Universal Robots PolyScope program: TurnToolFlange.urp

ProgramRoot directory=/home/ur/ursim-3.1/programs; kinematics=(a=[0, -0.425, -0.39225, 0, 0, 0], d=[0.08916, 0, 0, 0.10915, 0.09465, 0.0823], alpha=[1.5708, 0, 0, 1.5708, -1.5708, 0], deltaTheta=[0, 0, 0, 0, 0, 0], status=notInitialized); lastSavedInVersion=(project__name=Polyscope, major__version=3, minor__version=1, svn__revision=17195, build__date=Mar 11 2015, 13:02:28); name=TurnToolFlange; programVersion=(project__name=Polyscope, major__version=3, minor__version=1, svn__revision=17195, build__date=Mar 11 2015, 13:02:28); robotEnvironmentFileName=default; serialNumberRobot=2014350001
  MainProgram cartesianAcceleration=1.2; cartesianSpeed=0.25; jointAcceleration=1.3962634015954636; jointSpeed=1.0471975511965976; sharedProcessMoveBlendRadius=0.025; motionType=JOINT_SPACE; runOnlyOneCycle=true
    Move cartesianAcceleration=1.2; cartesianSpeed=0.25; jointAcceleration=1.3962634015954636; jointSpeed=1.0471975511965976; sharedProcessMoveBlendRadius=0.025; motionType=JOINT_SPACE
      Waypoint blendRadius=0.05; cartesianAcceleration=1.2; cartesianSpeed=0.25; jointAcceleration=1.3962634015954636; jointSpeed=1.0471975511965976; nextMotionTime=2.0; stoppoint=true; useSharedBlendParameter=true; useSharedParameters=true; outputFlangePose=(pos=(x=-0.12011316349511432, y=-0.4317629397815833, z=0.33440045381825007), rot=(x=-0.0012209830283371023, y=3.116276481240665, z=0.038891916168164946)); position=TCP in base x=-120.113 y=-431.763 z=334.4 mm, rx=-0.0012 ry=3.1163 rz=0.0389 rad; joints [-91.713, -84.826, -108.941, -77.706, 91.393, -1.776] deg; positionType=FIXED_POSITION; waypointPoseInFeatureCoordinates=(pos=(x=-0.12011316299633705, y=-0.4317629218220435, z=0.33440041081305716), rot=(x=-0.0012209830284087941, y=3.116276481240896, z=0.03889191616813282)); name=actual_pos
    Assignment expr=get_actual_joint_positions(); operatorValueType=INTEGER; valueSource=EXPRESSION
    Script type=0; expressionBranchNode=ExpressionVariableNode[5]=joint[5]+d2r(90)
    If checkConditionInSeperateThread=true; expr=ExpressionIONode≟ False; type=IF_NODE
      Move cartesianAcceleration=1.2; cartesianSpeed=0.25; jointAcceleration=1.3962634015954636; jointSpeed=1.0471975511965976; sharedProcessMoveBlendRadius=0.025; motionType=JOINT_SPACE
        Waypoint blendRadius=0.05; cartesianAcceleration=1.2; cartesianSpeed=0.25; jointAcceleration=1.3962634015954636; jointSpeed=1.0471975511965976; nextMotionTime=2.0; stoppoint=true; useSharedBlendParameter=true; useSharedParameters=true; positionType=VARIABLE_POSITION; name=Waypoint
    If type=ELSE_NODE
      Move cartesianAcceleration=1.2; cartesianSpeed=0.25; jointAcceleration=1.3962634015954636; jointSpeed=1.0471975511965976; sharedProcessMoveBlendRadius=0.025; motionType=JOINT_SPACE
        Waypoint blendRadius=0.05; cartesianAcceleration=1.2; cartesianSpeed=0.25; jointAcceleration=1.3962634015954636; jointSpeed=1.0471975511965976; nextMotionTime=2.0; stoppoint=true; useSharedBlendParameter=true; useSharedParameters=true; outputFlangePose=(pos=(x=-0.12011316349511432, y=-0.4317629397815833, z=0.33440045381825007), rot=(x=-0.0012209830283371023, y=3.116276481240665, z=0.038891916168164946)); position=TCP in base x=-120.113 y=-431.763 z=334.4 mm, rx=-0.0012 ry=3.1163 rz=0.0389 rad; joints [-91.713, -84.826, -108.941, -77.706, 91.393, -1.776] deg; positionType=FIXED_POSITION; waypointPoseInFeatureCoordinates=(pos=(x=-0.12011316299633705, y=-0.4317629218220435, z=0.33440041081305716), rot=(x=-0.0012209830284087941, y=3.116276481240896, z=0.03889191616813282)); name=actual_pos
